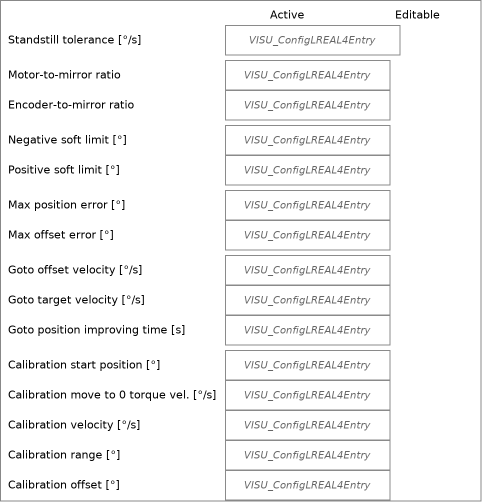
VISUALIZATION VISU_M3Config_Rotation_General  // 482x502
VAR_IN_OUT
	active : M3RotationConfig;
	editable : M3RotationConfig;
END_VAR
    Label (225,5 125x20), "Active"
    Label (355,5 125x20), "Editable"
    Label (5,25 140x30), "Standstill tolerance [°/s]"
    Frame (225,25 175x30)
        shows VISU_ConfigLREAL4Entry(active := active.standstillTolerance, editable := editable.standstillTolerance)
    Label (5,60 140x30), "Motor-to-mirror ratio"
    Frame (225,60 165x30)
        shows VISU_ConfigLREAL4Entry(active := active.motorToMirrorRatio, editable := editable.motorToMirrorRatio)
    Frame (225,90 165x30)
        shows VISU_ConfigLREAL4Entry(active := active.encoderToMirrorRatio, editable := editable.encoderToMirrorRatio)
    Label (5,90 140x30), "Encoder-to-mirror ratio"
    Label (5,125 140x30), "Negative soft limit [°]"
    Frame (225,125 165x30)
        shows VISU_ConfigLREAL4Entry(active := active.negativeSoftLimit, editable := editable.negativeSoftLimit)
    Frame (225,155 165x30)
        shows VISU_ConfigLREAL4Entry(active := active.positiveSoftLimit, editable := editable.positiveSoftLimit)
    Label (5,155 140x30), "Positive soft limit [°]"
    Label (5,190 140x30), "Max position error [°]"
    Frame (225,190 165x30)
        shows VISU_ConfigLREAL4Entry(active := active.maxPositionError, editable := editable.maxPositionError)
    Frame (225,220 165x30)
        shows VISU_ConfigLREAL4Entry(active := active.maxOffsetError, editable := editable.maxOffsetError)
    Label (5,220 140x30), "Max offset error [°]"
    Label (5,255 140x30), "Goto offset velocity [°/s]"
    Frame (225,255 165x30)
        shows VISU_ConfigLREAL4Entry(active := active.gotoOffsetVelocity, editable := editable.gotoOffsetVelocity)
    Label (5,315 180x30), "Goto position improving time [s]"
    Frame (225,285 165x30)
        shows VISU_ConfigLREAL4Entry(active := active.gotoTargetVelocity, editable := editable.gotoTargetVelocity)
    Label (5,285 140x30), "Goto target velocity [°/s]"
    Frame (225,315 165x30)
        shows VISU_ConfigLREAL4Entry(active := active.gotoImprovingPositionTime, editable := editable.gotoImprovingPositionTime)
    Frame (225,350 165x30)
        shows VISU_ConfigLREAL4Entry(active := active.calibrateStartPosition, editable := editable.calibrateStartPosition)
    Frame (225,380 165x30)
        shows VISU_ConfigLREAL4Entry(active := active.calibrateMoveToZeroTorqueVelocity, editable := editable.calibrateMoveToZeroTorqueVelocity)
    Frame (225,410 165x30)
        shows VISU_ConfigLREAL4Entry(active := active.calibrateVelocity, editable := editable.calibrateVelocity)
    Frame (225,440 165x30)
        shows VISU_ConfigLREAL4Entry(active := active.calibrateRange, editable := editable.calibrateRange)
    Frame (225,470 165x30)
        shows VISU_ConfigLREAL4Entry(active := active.calibrateOffset, editable := editable.calibrateOffset)
    Label (5,410 180x30), "Calibration velocity [°/s]"
    Label (5,350 185x30), "Calibration start position [°]"
    Label (5,380 235x30), "Calibration move to 0 torque vel. [°/s]"
    Label (5,470 140x30), "Calibration offset [°]"
    Label (5,440 140x30), "Calibration range [°]"
END_VISUALIZATION

(* stored: Version 1.1.0.1, ProductVersion 3.1.4019.2
   Visu VISU_M3Config_Rotation_General: Id {33f16c21-6e55-4f86-9cb4-d9f1af35d89b} *)
